FUNCTION F_CurveSpeed : LREAL
VAR_INPUT
END_VAR
VAR
END_VAR

END_FUNCTION

(* stored: Version 1.1.0.1, ProductVersion 3.1.0.25
   POU F_CurveSpeed: Id {4753b587-9e40-474c-b43b-c8cb78fcfddb} *)
